// TwinCAT 3 PLC project AdsAnyNetIdEx
// ProgramVersion: 3.1.4023.0
// libraries:
//   Tc2_DataExchange, * (Beckhoff Automation GmbH)
//   Tc2_Standard, * (Beckhoff Automation GmbH)
//   Tc2_System, * (Beckhoff Automation GmbH)
//   Tc2_Utilities, * (Beckhoff Automation GmbH)
//   Tc3_BA_Common, * (Beckhoff Automation GmbH)
//   Tc3_Module, * (Beckhoff Automation GmbH)
// project tree:
//   DUTs/ADS Package/ AdsData.TcDUT (not stored), AdsMessage.TcDUT (not stored), AdsMessageQueue.TcPOU (not stored), AdsSocket.TcPOU (not stored), Watchdog.TcPOU (not stored)
//   DUTs/ AreaNum.TcDUT (not stored), EventsEnum.TcTLEO (not stored)
//   GVLs/ Sockets.TcGVL (not stored)
//   / PlcTask.TcTTO (not stored)
//   POUs/ AdsTcpUnitEx.TcPOU, BufferIsEmpty.TcPOU (not stored), BytesToString.TcPOU (not stored), MAIN.TcPOU
// real-time tasks:
//   TASK PlcTask: cycle T#10ms, priority 21, ADS port 350

// ---- POUs/AdsTcpUnitEx.TcPOU
FUNCTION_BLOCK AdsTcpUnitEx
VAR_INPUT
	setMode : (SEND, QUEUE);
END_VAR
VAR_OUTPUT
	bBusy : BOOL;
	error : BOOL;
	errorID : UDINT;
END_VAR
VAR
	socketsArr : ARRAY[1..numSockets] OF POINTER TO AdsSocket; //use this to find a socket
	
	//declare all sockets here
	AREA_2 : AdsSocket := (PrgName := TO_STRING(AreaNum.AREA_2), AmsNetId := '', AmsPort := 851); //local socket, unused
	AREA_3 : AdsSocket := (PrgName := TO_STRING(AreaNum.AREA_3), AmsNetId := '3.0.131.216.1.1', AmsPort := 851); //placeholder NetId
END_VAR
VAR
	socket : REFERENCE TO AdsSocket;
	
	messageQueue : AdsMessageQueue;
	nextMessage : AdsMessage;
	
	mode : (SEND, QUEUE);
END_VAR
VAR CONSTANT
	numSockets : INT := 2;
END_VAR

(*
	this extended version of AdsTcp communication provides the option to dynamically generate ADS messages into a queue
		due to the significant stack memory requirements, the QUEUE model can only be used on systems with adjustable stack
		using QUEUE mode on panel PCs (CP66xx) or other mini controllers can freeze the system
		
	QUEUE mode:
		when a message is polled, a socket with the same recipient name is identified
			if the identified socket is ready to send, then the message is passed to the socket
			otherwise, the message is placed back into the queue
		if no socket with a matching name can be identified, then the message is discarded
		
	SEND mode:
		if a socket matching the recipient name is identified and it is not busy or in error state, then the message is passed
		
	sendMessage() specifies a recipient name and data contents, then checks the mode to determine how to handle the message
*)

fillSocketsArr();

IF messageQueue.isEmpty() THEN
	mode := setMode;
END_IF

blocks();

IF mode = QUEUE THEN
	pollAndSend();	
END_IF

METHOD PRIVATE blocks : BOOL
VAR_INPUT
END_VAR
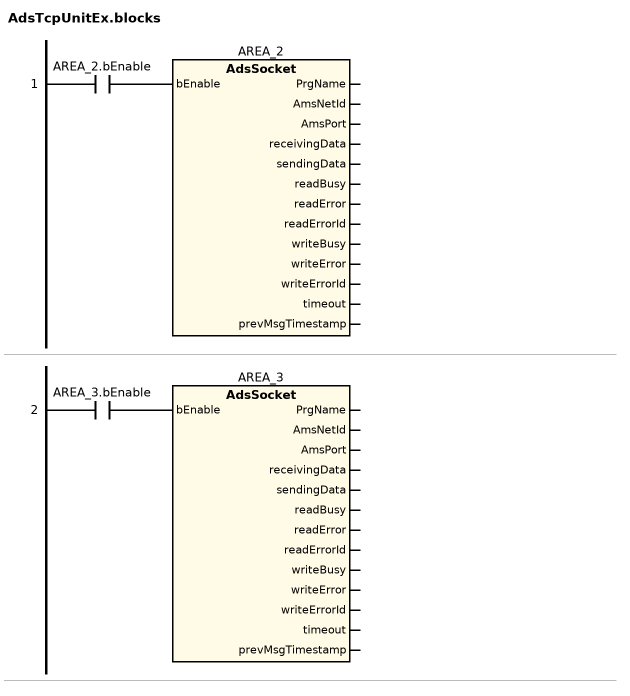
// NETWORK 1
AREA_2(bEnable := AREA_2.bEnable); // AdsSocket

// NETWORK 2
AREA_3(bEnable := AREA_3.bEnable); // AdsSocket
END_METHOD

METHOD fetchData : BOOL
VAR_INPUT
	senderName : STRING;
END_VAR
VAR_OUTPUT
	data : AdsData;
END_VAR
VAR
	i : INT;
END_VAR
FOR i:=1 TO numSockets BY 1 DO
	
	IF socketsArr[i]^.PrgName = senderName THEN
		fetchData := TRUE;
		data := socketsArr[i]^.receivingData;
		RETURN;
	END_IF
	
END_FOR
END_METHOD

METHOD PRIVATE fillSocketsArr : BOOL
VAR_INPUT
END_VAR
socketsArr[1] := ADR(AREA_2);
socketsArr[2] := ADR(AREA_3);
END_METHOD

METHOD PRIVATE findSocket : REFERENCE TO AdsSocket
VAR_INPUT
	recipient : STRING;
END_VAR
VAR
	i : INT;
END_VAR
FOR i:=1 TO numSockets BY 1 DO
	IF socketsArr[i] <> 0 AND_THEN socketsArr[i]^.PrgName = recipient THEN
		findSocket REF= socketsArr[i]^;
		RETURN;
	END_IF
END_FOR
END_METHOD

METHOD PRIVATE pollAndSend : BOOL
VAR_INPUT
END_VAR
nextMessage := messageQueue.poll(getSize => );
socket REF= findSocket(recipient := nextMessage.recipient);

IF __ISVALIDREF(socket) THEN
	
	IF NOT socket.writeBusy AND NOT socket.writeError AND socket.writeReady THEN
		socket.send(data := nextMessage.contents);
	ELSE //if socket is busy or has ERROR state, then message is returned to the end of the line
		messageQueue.push(value := nextMessage);
	END_IF
	
END_IF
END_METHOD

METHOD sendMessage : BOOL
VAR_INPUT
	recipient : STRING;
	data : REFERENCE TO AdsData;
END_VAR
VAR
	newMessage : AdsMessage;
END_VAR
CASE mode OF
	SEND:
		socket REF= findSocket(recipient := recipient);
		IF
			__ISVALIDREF(socket) AND_THEN
			NOT socket.writeBusy AND NOT socket.writeError
		THEN
			socket.send(data := data);
			sendMessage := TRUE;
		END_IF
	
	QUEUE:
		IF recipient <> '' THEN
			newMessage.recipient := recipient;
			newMessage.contents := data;
			
			sendMessage := messageQueue.push(newMessage);
		END_IF
	
END_CASE
END_METHOD

END_FUNCTION_BLOCK

// ---- POUs/MAIN.TcPOU
PROGRAM MAIN
VAR_OUTPUT
	localTime : TIMESTRUCT;
	year, month, day : WORD;
	hour, minute, second : WORD;
END_VAR
VAR
	sMessage : STRING := 'from AREA_4';
	newRecipient : STRING;
	newData : AdsData;
	retrievedData : AdsData;
	
	sendOnce : BOOL;
	sendFastNum : BOOL;
	
	i : INT := 0;
	
	fbLocalSystemTime : FB_LocalSystemTime;
END_VAR

readTime();	

blocks();
	
IF sendOnce OR sendFastNum THEN
	MEMSET(ADR(newData), 0, SIZEOF(newData));
	
	sMessage := TO_STRING(i);
	
	newRecipient := TO_STRING(AreaNum.AREA_4);
	newData.description := EventsEnum.TEST_COMMS;
	newData.timestamp := localTime;
	STRNCPY(ADR(newData.binaryData), ADR(sMessage), SIZEOF(sMessage));
	newData.binaryData[100000] := 69;
	
	IF
		adsMajorNetwork.sendMessage(recipient := newRecipient, data := newData)
	THEN
		i := i + 1;
		sendOnce := FALSE;
	END_IF	
END_IF

retrievedData := AREA_3.receivingData;

METHOD blocks : BOOL
VAR_INPUT
END_VAR
adsMajorNetwork(
	setMode:= 1, 
	bBusy=> , 
	error=> , 
	errorID=> );
	
adsLocalNetwork(
	setMode:= 1, 
	bBusy=> , 
	error=> , 
	errorID=> );
END_METHOD

METHOD readTime : BOOL
VAR_INPUT
END_VAR
fbLocalSystemTime(
	sNetID:= , 
	bEnable:= TRUE, 
	dwCycle:= , 
	dwOpt:= , 
	tTimeout:= , 
	bValid=> , 
	systemTime=> localTime, 
	tzID=> );
year := localTime.wYear;
month := localTime.wMonth;
day := localTime.wDay;
hour := localTime.wHour;
minute := localTime.wMinute;
second := localTime.wSecond;
END_METHOD

END_PROGRAM
